PROGRAM Vision
VAR
	VisionBase	: FB_VisionController;
	_ImageCount	: ULINT;
	ipImageResDisp	: ITcVnDisplayableImage;
END_VAR

VisionBase.CyclicLogic();

IF VisionBase.imageCount > _Imagecount THEN
	F_VN_CopyIntoDisplayableImage(VisionBase.ipImageIn, ipImageResDisp, VisionBase.hr);
END_IF

_ImageCount	:= VisionBase.imagecount;

END_PROGRAM

(* stored: Version 1.1.0.1
   POU Vision: Id {252271fb-6a71-407e-8f09-23cd75440a88}, SpecialFunc None *)
